{attribute 'qualified_only'}
{attribute 'strict'}
TYPE ActionMode :
(
	DoNothing	:= 0,
	AbsMove		:= 1,
	RelMove		:= 2,
	Home		:= 3,
	Find		:= 4
);
END_TYPE

(* stored: Version 1.1.0.1, ProductVersion 3.1.4024.14
   DUT ActionMode: Id {36e4c4f3-2e63-4aad-9522-c77b711e5f9d} *)
